(* IEC 61131-3 sources: TIA2AX/tests/test_projects/expected/HW_2200330_V18/ST70_PLC, 6 files *)

(* ---- HwInputs.st ---- *)
TYPE
	HwInputs : STRUCT
		ST70_ET200SP_CM_4xIO_Link_1 AT %B100 : ARRAY[0..31] OF BYTE;
		ST70_ET200SP_DI_16x24VDC_ST_1 AT %B0 : WORD;
		ST70_ET200SP_DI_16x24VDC_ST_2 AT %B2 : WORD;
		ST70_ET200SP_DI_8x24VDC_ST_3 AT %B4 : BYTE;
		ST70_ET200SP_DI_16x24VDC_ST_4 AT %B5 : WORD;
		ST70_1_DM260_PB_Acquisition_Status_1 AT %B1000 : ARRAY[0..2] OF BYTE;
		ST70_1_DM260_PB_Results_Status_1 AT %B1003 : BYTE;
		ST70_1_DM260_PB_Soft_Event_Control_1 AT %B1004 : BYTE;
		ST70_1_DM260_PB_Result_Data_64_bytes_1 AT %B1010 : ARRAY[0..71] OF BYTE;
		ST70_2_DM260_PB_Acquisition_Status_1 AT %B2000 : ARRAY[0..2] OF BYTE;
		ST70_2_DM260_PB_Results_Status_1 AT %B2003 : BYTE;
		ST70_2_DM260_PB_Soft_Event_Control_1 AT %B2004 : BYTE;
		ST70_2_DM260_PB_Result_Data_64_bytes_1 AT %B2010 : ARRAY[0..71] OF BYTE;
		ST70_3_DM260_PB_Acquisition_Status_1 AT %B3000 : ARRAY[0..2] OF BYTE;
		ST70_3_DM260_PB_Results_Status_1 AT %B3003 : BYTE;
		ST70_3_DM260_PB_Soft_Event_Control_1 AT %B3004 : BYTE;
		ST70_3_DM260_PB_Result_Data_64_bytes_1 AT %B3010 : ARRAY[0..71] OF BYTE;
		ST70_1_DM260_EB_Acquisition_Status_1 AT %B1200 : ARRAY[0..2] OF BYTE;
		ST70_1_DM260_EB_Results_Status_1 AT %B1203 : BYTE;
		ST70_1_DM260_EB_Soft_Event_Control_1 AT %B1204 : BYTE;
		ST70_1_DM260_EB_Result_Data_64_bytes_1 AT %B1210 : ARRAY[0..71] OF BYTE;
		ST70_2_DM260_EB_Acquisition_Status_1 AT %B2200 : ARRAY[0..2] OF BYTE;
		ST70_2_DM260_EB_Results_Status_1 AT %B2203 : BYTE;
		ST70_2_DM260_EB_Soft_Event_Control_1 AT %B2204 : BYTE;
		ST70_2_DM260_EB_Result_Data_64_bytes_1 AT %B2210 : ARRAY[0..71] OF BYTE;
		ST70_3_DM260_EB_Acquisition_Status_1 AT %B3200 : ARRAY[0..2] OF BYTE;
		ST70_3_DM260_EB_Results_Status_1 AT %B3203 : BYTE;
		ST70_3_DM260_EB_Soft_Event_Control_1 AT %B3204 : BYTE;
		ST70_3_DM260_EB_Result_Data_64_bytes_1 AT %B3210 : ARRAY[0..71] OF BYTE;
	END_STRUCT;
END_TYPE

(* ---- HwOutputs.st ---- *)
TYPE
	HwOutputs : STRUCT
		ST70_ET200SP_CM_4xIO_Link_1 AT %B100 : ARRAY[0..31] OF BYTE;
		ST70_ET200SP_DQ_16x24VDC_0_5A_ST_1 AT %B0 : WORD;
		ST70_ET200SP_DQ_16x24VDC_0_5A_ST_2 AT %B2 : WORD;
		ST70_ET200SP_DQ_16x24VDC_0_5A_ST_3 AT %B4 : WORD;
		ST70_CPX_MPA1S_VMPA1_FB_EMS_8_8DO_1 AT %B200 : BYTE;
		ST70_CPX_MPA1S_VMPA1_FB_EMS_8_8DO_2 AT %B201 : BYTE;
		ST70_CPX_MPA1S_VMPA1_FB_EMS_8_8DO_3 AT %B202 : BYTE;
		ST70_CPX_MPA2S_VMPA2_FB_EMS_4_4DO_1 AT %B6 : BYTE;
		ST70_CPX_MPA1G_VMPA1_FB_EMG_8_8DO_3 AT %B204 : BYTE;
		ST70_1_DM260_PB_Acquisition_Control_1 AT %B1000 : BYTE;
		ST70_1_DM260_PB_Results_Control_1 AT %B1003 : BYTE;
		ST70_1_DM260_PB_Soft_Event_Control_1 AT %B1004 : BYTE;
		ST70_1_DM260_PB_User_Data_64_bytes_1 AT %B1010 : ARRAY[0..67] OF BYTE;
		ST70_2_DM260_PB_Acquisition_Control_1 AT %B2000 : BYTE;
		ST70_2_DM260_PB_Results_Control_1 AT %B2003 : BYTE;
		ST70_2_DM260_PB_Soft_Event_Control_1 AT %B2004 : BYTE;
		ST70_2_DM260_PB_User_Data_64_bytes_1 AT %B2010 : ARRAY[0..67] OF BYTE;
		ST70_3_DM260_PB_Acquisition_Control_1 AT %B3000 : BYTE;
		ST70_3_DM260_PB_Results_Control_1 AT %B3003 : BYTE;
		ST70_3_DM260_PB_Soft_Event_Control_1 AT %B3004 : BYTE;
		ST70_3_DM260_PB_User_Data_64_bytes_1 AT %B3010 : ARRAY[0..67] OF BYTE;
		ST70_1_DM260_EB_Acquisition_Control_1 AT %B1200 : BYTE;
		ST70_1_DM260_EB_Results_Control_1 AT %B1203 : BYTE;
		ST70_1_DM260_EB_Soft_Event_Control_1 AT %B1204 : BYTE;
		ST70_1_DM260_EB_User_Data_64_bytes_1 AT %B1210 : ARRAY[0..67] OF BYTE;
		ST70_2_DM260_EB_Acquisition_Control_1 AT %B2200 : BYTE;
		ST70_2_DM260_EB_Results_Control_1 AT %B2203 : BYTE;
		ST70_2_DM260_EB_Soft_Event_Control_1 AT %B2204 : BYTE;
		ST70_2_DM260_EB_User_Data_64_bytes_1 AT %B2210 : ARRAY[0..67] OF BYTE;
		ST70_3_DM260_EB_Acquisition_Control_1 AT %B3200 : BYTE;
		ST70_3_DM260_EB_Results_Control_1 AT %B3203 : BYTE;
		ST70_3_DM260_EB_Soft_Event_Control_1 AT %B3204 : BYTE;
		ST70_3_DM260_EB_User_Data_64_bytes_1 AT %B3210 : ARRAY[0..67] OF BYTE;
	END_STRUCT;
END_TYPE

(* ---- PlcInputs.st ---- *)
TYPE
	PlcInputs : STRUCT
		ST70_ET200SP_CM_4xIO_Link_1 : ARRAY[0..31] OF BYTE;
		ST70_ET200SP_DI_16x24VDC_ST_1 : WORD;
		ST70_ET200SP_DI_16x24VDC_ST_2 : WORD;
		ST70_ET200SP_DI_8x24VDC_ST_3 : BYTE;
		ST70_ET200SP_DI_16x24VDC_ST_4 : WORD;
		ST70_1_DM260_PB_Acquisition_Status_1 : ARRAY[0..2] OF BYTE;
		ST70_1_DM260_PB_Results_Status_1 : BYTE;
		ST70_1_DM260_PB_Soft_Event_Control_1 : BYTE;
		ST70_1_DM260_PB_Result_Data_64_bytes_1 : ARRAY[0..71] OF BYTE;
		ST70_2_DM260_PB_Acquisition_Status_1 : ARRAY[0..2] OF BYTE;
		ST70_2_DM260_PB_Results_Status_1 : BYTE;
		ST70_2_DM260_PB_Soft_Event_Control_1 : BYTE;
		ST70_2_DM260_PB_Result_Data_64_bytes_1 : ARRAY[0..71] OF BYTE;
		ST70_3_DM260_PB_Acquisition_Status_1 : ARRAY[0..2] OF BYTE;
		ST70_3_DM260_PB_Results_Status_1 : BYTE;
		ST70_3_DM260_PB_Soft_Event_Control_1 : BYTE;
		ST70_3_DM260_PB_Result_Data_64_bytes_1 : ARRAY[0..71] OF BYTE;
		ST70_1_DM260_EB_Acquisition_Status_1 : ARRAY[0..2] OF BYTE;
		ST70_1_DM260_EB_Results_Status_1 : BYTE;
		ST70_1_DM260_EB_Soft_Event_Control_1 : BYTE;
		ST70_1_DM260_EB_Result_Data_64_bytes_1 : ARRAY[0..71] OF BYTE;
		ST70_2_DM260_EB_Acquisition_Status_1 : ARRAY[0..2] OF BYTE;
		ST70_2_DM260_EB_Results_Status_1 : BYTE;
		ST70_2_DM260_EB_Soft_Event_Control_1 : BYTE;
		ST70_2_DM260_EB_Result_Data_64_bytes_1 : ARRAY[0..71] OF BYTE;
		ST70_3_DM260_EB_Acquisition_Status_1 : ARRAY[0..2] OF BYTE;
		ST70_3_DM260_EB_Results_Status_1 : BYTE;
		ST70_3_DM260_EB_Soft_Event_Control_1 : BYTE;
		ST70_3_DM260_EB_Result_Data_64_bytes_1 : ARRAY[0..71] OF BYTE;
	END_STRUCT;
END_TYPE

(* ---- PlcOutputs.st ---- *)
TYPE
	PlcOutputs : STRUCT
		ST70_ET200SP_CM_4xIO_Link_1 : ARRAY[0..31] OF BYTE;
		ST70_ET200SP_DQ_16x24VDC_0_5A_ST_1 : WORD;
		ST70_ET200SP_DQ_16x24VDC_0_5A_ST_2 : WORD;
		ST70_ET200SP_DQ_16x24VDC_0_5A_ST_3 : WORD;
		ST70_CPX_MPA1S_VMPA1_FB_EMS_8_8DO_1 : BYTE;
		ST70_CPX_MPA1S_VMPA1_FB_EMS_8_8DO_2 : BYTE;
		ST70_CPX_MPA1S_VMPA1_FB_EMS_8_8DO_3 : BYTE;
		ST70_CPX_MPA2S_VMPA2_FB_EMS_4_4DO_1 : BYTE;
		ST70_CPX_MPA1G_VMPA1_FB_EMG_8_8DO_3 : BYTE;
		ST70_1_DM260_PB_Acquisition_Control_1 : BYTE;
		ST70_1_DM260_PB_Results_Control_1 : BYTE;
		ST70_1_DM260_PB_Soft_Event_Control_1 : BYTE;
		ST70_1_DM260_PB_User_Data_64_bytes_1 : ARRAY[0..67] OF BYTE;
		ST70_2_DM260_PB_Acquisition_Control_1 : BYTE;
		ST70_2_DM260_PB_Results_Control_1 : BYTE;
		ST70_2_DM260_PB_Soft_Event_Control_1 : BYTE;
		ST70_2_DM260_PB_User_Data_64_bytes_1 : ARRAY[0..67] OF BYTE;
		ST70_3_DM260_PB_Acquisition_Control_1 : BYTE;
		ST70_3_DM260_PB_Results_Control_1 : BYTE;
		ST70_3_DM260_PB_Soft_Event_Control_1 : BYTE;
		ST70_3_DM260_PB_User_Data_64_bytes_1 : ARRAY[0..67] OF BYTE;
		ST70_1_DM260_EB_Acquisition_Control_1 : BYTE;
		ST70_1_DM260_EB_Results_Control_1 : BYTE;
		ST70_1_DM260_EB_Soft_Event_Control_1 : BYTE;
		ST70_1_DM260_EB_User_Data_64_bytes_1 : ARRAY[0..67] OF BYTE;
		ST70_2_DM260_EB_Acquisition_Control_1 : BYTE;
		ST70_2_DM260_EB_Results_Control_1 : BYTE;
		ST70_2_DM260_EB_Soft_Event_Control_1 : BYTE;
		ST70_2_DM260_EB_User_Data_64_bytes_1 : ARRAY[0..67] OF BYTE;
		ST70_3_DM260_EB_Acquisition_Control_1 : BYTE;
		ST70_3_DM260_EB_Results_Control_1 : BYTE;
		ST70_3_DM260_EB_Soft_Event_Control_1 : BYTE;
		ST70_3_DM260_EB_User_Data_64_bytes_1 : ARRAY[0..67] OF BYTE;
	END_STRUCT;
END_TYPE

(* ---- CopyInputs.st ---- *)
FUNCTION CopyInputs
	VAR_EXTERNAL
		HwInputs : HwInputs;
		PlcInputs : PlcInputs;
	END_VAR
	PlcInputs.ST70_ET200SP_CM_4xIO_Link_1[0] := HwInputs.ST70_ET200SP_CM_4xIO_Link_1[0];
	PlcInputs.ST70_ET200SP_CM_4xIO_Link_1[1] := HwInputs.ST70_ET200SP_CM_4xIO_Link_1[1];
	PlcInputs.ST70_ET200SP_CM_4xIO_Link_1[2] := HwInputs.ST70_ET200SP_CM_4xIO_Link_1[2];
	PlcInputs.ST70_ET200SP_CM_4xIO_Link_1[3] := HwInputs.ST70_ET200SP_CM_4xIO_Link_1[3];
	PlcInputs.ST70_ET200SP_CM_4xIO_Link_1[4] := HwInputs.ST70_ET200SP_CM_4xIO_Link_1[4];
	PlcInputs.ST70_ET200SP_CM_4xIO_Link_1[5] := HwInputs.ST70_ET200SP_CM_4xIO_Link_1[5];
	PlcInputs.ST70_ET200SP_CM_4xIO_Link_1[6] := HwInputs.ST70_ET200SP_CM_4xIO_Link_1[6];
	PlcInputs.ST70_ET200SP_CM_4xIO_Link_1[7] := HwInputs.ST70_ET200SP_CM_4xIO_Link_1[7];
	PlcInputs.ST70_ET200SP_CM_4xIO_Link_1[8] := HwInputs.ST70_ET200SP_CM_4xIO_Link_1[8];
	PlcInputs.ST70_ET200SP_CM_4xIO_Link_1[9] := HwInputs.ST70_ET200SP_CM_4xIO_Link_1[9];
	PlcInputs.ST70_ET200SP_CM_4xIO_Link_1[10] := HwInputs.ST70_ET200SP_CM_4xIO_Link_1[10];
	PlcInputs.ST70_ET200SP_CM_4xIO_Link_1[11] := HwInputs.ST70_ET200SP_CM_4xIO_Link_1[11];
	PlcInputs.ST70_ET200SP_CM_4xIO_Link_1[12] := HwInputs.ST70_ET200SP_CM_4xIO_Link_1[12];
	PlcInputs.ST70_ET200SP_CM_4xIO_Link_1[13] := HwInputs.ST70_ET200SP_CM_4xIO_Link_1[13];
	PlcInputs.ST70_ET200SP_CM_4xIO_Link_1[14] := HwInputs.ST70_ET200SP_CM_4xIO_Link_1[14];
	PlcInputs.ST70_ET200SP_CM_4xIO_Link_1[15] := HwInputs.ST70_ET200SP_CM_4xIO_Link_1[15];
	PlcInputs.ST70_ET200SP_CM_4xIO_Link_1[16] := HwInputs.ST70_ET200SP_CM_4xIO_Link_1[16];
	PlcInputs.ST70_ET200SP_CM_4xIO_Link_1[17] := HwInputs.ST70_ET200SP_CM_4xIO_Link_1[17];
	PlcInputs.ST70_ET200SP_CM_4xIO_Link_1[18] := HwInputs.ST70_ET200SP_CM_4xIO_Link_1[18];
	PlcInputs.ST70_ET200SP_CM_4xIO_Link_1[19] := HwInputs.ST70_ET200SP_CM_4xIO_Link_1[19];
	PlcInputs.ST70_ET200SP_CM_4xIO_Link_1[20] := HwInputs.ST70_ET200SP_CM_4xIO_Link_1[20];
	PlcInputs.ST70_ET200SP_CM_4xIO_Link_1[21] := HwInputs.ST70_ET200SP_CM_4xIO_Link_1[21];
	PlcInputs.ST70_ET200SP_CM_4xIO_Link_1[22] := HwInputs.ST70_ET200SP_CM_4xIO_Link_1[22];
	PlcInputs.ST70_ET200SP_CM_4xIO_Link_1[23] := HwInputs.ST70_ET200SP_CM_4xIO_Link_1[23];
	PlcInputs.ST70_ET200SP_CM_4xIO_Link_1[24] := HwInputs.ST70_ET200SP_CM_4xIO_Link_1[24];
	PlcInputs.ST70_ET200SP_CM_4xIO_Link_1[25] := HwInputs.ST70_ET200SP_CM_4xIO_Link_1[25];
	PlcInputs.ST70_ET200SP_CM_4xIO_Link_1[26] := HwInputs.ST70_ET200SP_CM_4xIO_Link_1[26];
	PlcInputs.ST70_ET200SP_CM_4xIO_Link_1[27] := HwInputs.ST70_ET200SP_CM_4xIO_Link_1[27];
	PlcInputs.ST70_ET200SP_CM_4xIO_Link_1[28] := HwInputs.ST70_ET200SP_CM_4xIO_Link_1[28];
	PlcInputs.ST70_ET200SP_CM_4xIO_Link_1[29] := HwInputs.ST70_ET200SP_CM_4xIO_Link_1[29];
	PlcInputs.ST70_ET200SP_CM_4xIO_Link_1[30] := HwInputs.ST70_ET200SP_CM_4xIO_Link_1[30];
	PlcInputs.ST70_ET200SP_CM_4xIO_Link_1[31] := HwInputs.ST70_ET200SP_CM_4xIO_Link_1[31];
	PlcInputs.ST70_ET200SP_DI_16x24VDC_ST_1 := HwInputs.ST70_ET200SP_DI_16x24VDC_ST_1;
	PlcInputs.ST70_ET200SP_DI_16x24VDC_ST_2 := HwInputs.ST70_ET200SP_DI_16x24VDC_ST_2;
	PlcInputs.ST70_ET200SP_DI_8x24VDC_ST_3 := HwInputs.ST70_ET200SP_DI_8x24VDC_ST_3;
	PlcInputs.ST70_ET200SP_DI_16x24VDC_ST_4 := HwInputs.ST70_ET200SP_DI_16x24VDC_ST_4;
	PlcInputs.ST70_1_DM260_PB_Acquisition_Status_1[0] := HwInputs.ST70_1_DM260_PB_Acquisition_Status_1[0];
	PlcInputs.ST70_1_DM260_PB_Acquisition_Status_1[1] := HwInputs.ST70_1_DM260_PB_Acquisition_Status_1[1];
	PlcInputs.ST70_1_DM260_PB_Acquisition_Status_1[2] := HwInputs.ST70_1_DM260_PB_Acquisition_Status_1[2];
	PlcInputs.ST70_1_DM260_PB_Results_Status_1 := HwInputs.ST70_1_DM260_PB_Results_Status_1;
	PlcInputs.ST70_1_DM260_PB_Soft_Event_Control_1 := HwInputs.ST70_1_DM260_PB_Soft_Event_Control_1;
	PlcInputs.ST70_1_DM260_PB_Result_Data_64_bytes_1[0] := HwInputs.ST70_1_DM260_PB_Result_Data_64_bytes_1[0];
	PlcInputs.ST70_1_DM260_PB_Result_Data_64_bytes_1[1] := HwInputs.ST70_1_DM260_PB_Result_Data_64_bytes_1[1];
	PlcInputs.ST70_1_DM260_PB_Result_Data_64_bytes_1[2] := HwInputs.ST70_1_DM260_PB_Result_Data_64_bytes_1[2];
	PlcInputs.ST70_1_DM260_PB_Result_Data_64_bytes_1[3] := HwInputs.ST70_1_DM260_PB_Result_Data_64_bytes_1[3];
	PlcInputs.ST70_1_DM260_PB_Result_Data_64_bytes_1[4] := HwInputs.ST70_1_DM260_PB_Result_Data_64_bytes_1[4];
	PlcInputs.ST70_1_DM260_PB_Result_Data_64_bytes_1[5] := HwInputs.ST70_1_DM260_PB_Result_Data_64_bytes_1[5];
	PlcInputs.ST70_1_DM260_PB_Result_Data_64_bytes_1[6] := HwInputs.ST70_1_DM260_PB_Result_Data_64_bytes_1[6];
	PlcInputs.ST70_1_DM260_PB_Result_Data_64_bytes_1[7] := HwInputs.ST70_1_DM260_PB_Result_Data_64_bytes_1[7];
	PlcInputs.ST70_1_DM260_PB_Result_Data_64_bytes_1[8] := HwInputs.ST70_1_DM260_PB_Result_Data_64_bytes_1[8];
	PlcInputs.ST70_1_DM260_PB_Result_Data_64_bytes_1[9] := HwInputs.ST70_1_DM260_PB_Result_Data_64_bytes_1[9];
	PlcInputs.ST70_1_DM260_PB_Result_Data_64_bytes_1[10] := HwInputs.ST70_1_DM260_PB_Result_Data_64_bytes_1[10];
	PlcInputs.ST70_1_DM260_PB_Result_Data_64_bytes_1[11] := HwInputs.ST70_1_DM260_PB_Result_Data_64_bytes_1[11];
	PlcInputs.ST70_1_DM260_PB_Result_Data_64_bytes_1[12] := HwInputs.ST70_1_DM260_PB_Result_Data_64_bytes_1[12];
	PlcInputs.ST70_1_DM260_PB_Result_Data_64_bytes_1[13] := HwInputs.ST70_1_DM260_PB_Result_Data_64_bytes_1[13];
	PlcInputs.ST70_1_DM260_PB_Result_Data_64_bytes_1[14] := HwInputs.ST70_1_DM260_PB_Result_Data_64_bytes_1[14];
	PlcInputs.ST70_1_DM260_PB_Result_Data_64_bytes_1[15] := HwInputs.ST70_1_DM260_PB_Result_Data_64_bytes_1[15];
	PlcInputs.ST70_1_DM260_PB_Result_Data_64_bytes_1[16] := HwInputs.ST70_1_DM260_PB_Result_Data_64_bytes_1[16];
	PlcInputs.ST70_1_DM260_PB_Result_Data_64_bytes_1[17] := HwInputs.ST70_1_DM260_PB_Result_Data_64_bytes_1[17];
	PlcInputs.ST70_1_DM260_PB_Result_Data_64_bytes_1[18] := HwInputs.ST70_1_DM260_PB_Result_Data_64_bytes_1[18];
	PlcInputs.ST70_1_DM260_PB_Result_Data_64_bytes_1[19] := HwInputs.ST70_1_DM260_PB_Result_Data_64_bytes_1[19];
	PlcInputs.ST70_1_DM260_PB_Result_Data_64_bytes_1[20] := HwInputs.ST70_1_DM260_PB_Result_Data_64_bytes_1[20];
	PlcInputs.ST70_1_DM260_PB_Result_Data_64_bytes_1[21] := HwInputs.ST70_1_DM260_PB_Result_Data_64_bytes_1[21];
	PlcInputs.ST70_1_DM260_PB_Result_Data_64_bytes_1[22] := HwInputs.ST70_1_DM260_PB_Result_Data_64_bytes_1[22];
	PlcInputs.ST70_1_DM260_PB_Result_Data_64_bytes_1[23] := HwInputs.ST70_1_DM260_PB_Result_Data_64_bytes_1[23];
	PlcInputs.ST70_1_DM260_PB_Result_Data_64_bytes_1[24] := HwInputs.ST70_1_DM260_PB_Result_Data_64_bytes_1[24];
	PlcInputs.ST70_1_DM260_PB_Result_Data_64_bytes_1[25] := HwInputs.ST70_1_DM260_PB_Result_Data_64_bytes_1[25];
	PlcInputs.ST70_1_DM260_PB_Result_Data_64_bytes_1[26] := HwInputs.ST70_1_DM260_PB_Result_Data_64_bytes_1[26];
	PlcInputs.ST70_1_DM260_PB_Result_Data_64_bytes_1[27] := HwInputs.ST70_1_DM260_PB_Result_Data_64_bytes_1[27];
	PlcInputs.ST70_1_DM260_PB_Result_Data_64_bytes_1[28] := HwInputs.ST70_1_DM260_PB_Result_Data_64_bytes_1[28];
	PlcInputs.ST70_1_DM260_PB_Result_Data_64_bytes_1[29] := HwInputs.ST70_1_DM260_PB_Result_Data_64_bytes_1[29];
	PlcInputs.ST70_1_DM260_PB_Result_Data_64_bytes_1[30] := HwInputs.ST70_1_DM260_PB_Result_Data_64_bytes_1[30];
	PlcInputs.ST70_1_DM260_PB_Result_Data_64_bytes_1[31] := HwInputs.ST70_1_DM260_PB_Result_Data_64_bytes_1[31];
	PlcInputs.ST70_1_DM260_PB_Result_Data_64_bytes_1[32] := HwInputs.ST70_1_DM260_PB_Result_Data_64_bytes_1[32];
	PlcInputs.ST70_1_DM260_PB_Result_Data_64_bytes_1[33] := HwInputs.ST70_1_DM260_PB_Result_Data_64_bytes_1[33];
	PlcInputs.ST70_1_DM260_PB_Result_Data_64_bytes_1[34] := HwInputs.ST70_1_DM260_PB_Result_Data_64_bytes_1[34];
	PlcInputs.ST70_1_DM260_PB_Result_Data_64_bytes_1[35] := HwInputs.ST70_1_DM260_PB_Result_Data_64_bytes_1[35];
	PlcInputs.ST70_1_DM260_PB_Result_Data_64_bytes_1[36] := HwInputs.ST70_1_DM260_PB_Result_Data_64_bytes_1[36];
	PlcInputs.ST70_1_DM260_PB_Result_Data_64_bytes_1[37] := HwInputs.ST70_1_DM260_PB_Result_Data_64_bytes_1[37];
	PlcInputs.ST70_1_DM260_PB_Result_Data_64_bytes_1[38] := HwInputs.ST70_1_DM260_PB_Result_Data_64_bytes_1[38];
	PlcInputs.ST70_1_DM260_PB_Result_Data_64_bytes_1[39] := HwInputs.ST70_1_DM260_PB_Result_Data_64_bytes_1[39];
	PlcInputs.ST70_1_DM260_PB_Result_Data_64_bytes_1[40] := HwInputs.ST70_1_DM260_PB_Result_Data_64_bytes_1[40];
	PlcInputs.ST70_1_DM260_PB_Result_Data_64_bytes_1[41] := HwInputs.ST70_1_DM260_PB_Result_Data_64_bytes_1[41];
	PlcInputs.ST70_1_DM260_PB_Result_Data_64_bytes_1[42] := HwInputs.ST70_1_DM260_PB_Result_Data_64_bytes_1[42];
	PlcInputs.ST70_1_DM260_PB_Result_Data_64_bytes_1[43] := HwInputs.ST70_1_DM260_PB_Result_Data_64_bytes_1[43];
	PlcInputs.ST70_1_DM260_PB_Result_Data_64_bytes_1[44] := HwInputs.ST70_1_DM260_PB_Result_Data_64_bytes_1[44];
	PlcInputs.ST70_1_DM260_PB_Result_Data_64_bytes_1[45] := HwInputs.ST70_1_DM260_PB_Result_Data_64_bytes_1[45];
	PlcInputs.ST70_1_DM260_PB_Result_Data_64_bytes_1[46] := HwInputs.ST70_1_DM260_PB_Result_Data_64_bytes_1[46];
	PlcInputs.ST70_1_DM260_PB_Result_Data_64_bytes_1[47] := HwInputs.ST70_1_DM260_PB_Result_Data_64_bytes_1[47];
	PlcInputs.ST70_1_DM260_PB_Result_Data_64_bytes_1[48] := HwInputs.ST70_1_DM260_PB_Result_Data_64_bytes_1[48];
	PlcInputs.ST70_1_DM260_PB_Result_Data_64_bytes_1[49] := HwInputs.ST70_1_DM260_PB_Result_Data_64_bytes_1[49];
	PlcInputs.ST70_1_DM260_PB_Result_Data_64_bytes_1[50] := HwInputs.ST70_1_DM260_PB_Result_Data_64_bytes_1[50];
	PlcInputs.ST70_1_DM260_PB_Result_Data_64_bytes_1[51] := HwInputs.ST70_1_DM260_PB_Result_Data_64_bytes_1[51];
	PlcInputs.ST70_1_DM260_PB_Result_Data_64_bytes_1[52] := HwInputs.ST70_1_DM260_PB_Result_Data_64_bytes_1[52];
	PlcInputs.ST70_1_DM260_PB_Result_Data_64_bytes_1[53] := HwInputs.ST70_1_DM260_PB_Result_Data_64_bytes_1[53];
	PlcInputs.ST70_1_DM260_PB_Result_Data_64_bytes_1[54] := HwInputs.ST70_1_DM260_PB_Result_Data_64_bytes_1[54];
	PlcInputs.ST70_1_DM260_PB_Result_Data_64_bytes_1[55] := HwInputs.ST70_1_DM260_PB_Result_Data_64_bytes_1[55];
	PlcInputs.ST70_1_DM260_PB_Result_Data_64_bytes_1[56] := HwInputs.ST70_1_DM260_PB_Result_Data_64_bytes_1[56];
	PlcInputs.ST70_1_DM260_PB_Result_Data_64_bytes_1[57] := HwInputs.ST70_1_DM260_PB_Result_Data_64_bytes_1[57];
	PlcInputs.ST70_1_DM260_PB_Result_Data_64_bytes_1[58] := HwInputs.ST70_1_DM260_PB_Result_Data_64_bytes_1[58];
	PlcInputs.ST70_1_DM260_PB_Result_Data_64_bytes_1[59] := HwInputs.ST70_1_DM260_PB_Result_Data_64_bytes_1[59];
	PlcInputs.ST70_1_DM260_PB_Result_Data_64_bytes_1[60] := HwInputs.ST70_1_DM260_PB_Result_Data_64_bytes_1[60];
	PlcInputs.ST70_1_DM260_PB_Result_Data_64_bytes_1[61] := HwInputs.ST70_1_DM260_PB_Result_Data_64_bytes_1[61];
	PlcInputs.ST70_1_DM260_PB_Result_Data_64_bytes_1[62] := HwInputs.ST70_1_DM260_PB_Result_Data_64_bytes_1[62];
	PlcInputs.ST70_1_DM260_PB_Result_Data_64_bytes_1[63] := HwInputs.ST70_1_DM260_PB_Result_Data_64_bytes_1[63];
	PlcInputs.ST70_1_DM260_PB_Result_Data_64_bytes_1[64] := HwInputs.ST70_1_DM260_PB_Result_Data_64_bytes_1[64];
	PlcInputs.ST70_1_DM260_PB_Result_Data_64_bytes_1[65] := HwInputs.ST70_1_DM260_PB_Result_Data_64_bytes_1[65];
	PlcInputs.ST70_1_DM260_PB_Result_Data_64_bytes_1[66] := HwInputs.ST70_1_DM260_PB_Result_Data_64_bytes_1[66];
	PlcInputs.ST70_1_DM260_PB_Result_Data_64_bytes_1[67] := HwInputs.ST70_1_DM260_PB_Result_Data_64_bytes_1[67];
	PlcInputs.ST70_1_DM260_PB_Result_Data_64_bytes_1[68] := HwInputs.ST70_1_DM260_PB_Result_Data_64_bytes_1[68];
	PlcInputs.ST70_1_DM260_PB_Result_Data_64_bytes_1[69] := HwInputs.ST70_1_DM260_PB_Result_Data_64_bytes_1[69];
	PlcInputs.ST70_1_DM260_PB_Result_Data_64_bytes_1[70] := HwInputs.ST70_1_DM260_PB_Result_Data_64_bytes_1[70];
	PlcInputs.ST70_1_DM260_PB_Result_Data_64_bytes_1[71] := HwInputs.ST70_1_DM260_PB_Result_Data_64_bytes_1[71];
	PlcInputs.ST70_2_DM260_PB_Acquisition_Status_1[0] := HwInputs.ST70_2_DM260_PB_Acquisition_Status_1[0];
	PlcInputs.ST70_2_DM260_PB_Acquisition_Status_1[1] := HwInputs.ST70_2_DM260_PB_Acquisition_Status_1[1];
	PlcInputs.ST70_2_DM260_PB_Acquisition_Status_1[2] := HwInputs.ST70_2_DM260_PB_Acquisition_Status_1[2];
	PlcInputs.ST70_2_DM260_PB_Results_Status_1 := HwInputs.ST70_2_DM260_PB_Results_Status_1;
	PlcInputs.ST70_2_DM260_PB_Soft_Event_Control_1 := HwInputs.ST70_2_DM260_PB_Soft_Event_Control_1;
	PlcInputs.ST70_2_DM260_PB_Result_Data_64_bytes_1[0] := HwInputs.ST70_2_DM260_PB_Result_Data_64_bytes_1[0];
	PlcInputs.ST70_2_DM260_PB_Result_Data_64_bytes_1[1] := HwInputs.ST70_2_DM260_PB_Result_Data_64_bytes_1[1];
	PlcInputs.ST70_2_DM260_PB_Result_Data_64_bytes_1[2] := HwInputs.ST70_2_DM260_PB_Result_Data_64_bytes_1[2];
	PlcInputs.ST70_2_DM260_PB_Result_Data_64_bytes_1[3] := HwInputs.ST70_2_DM260_PB_Result_Data_64_bytes_1[3];
	PlcInputs.ST70_2_DM260_PB_Result_Data_64_bytes_1[4] := HwInputs.ST70_2_DM260_PB_Result_Data_64_bytes_1[4];
	PlcInputs.ST70_2_DM260_PB_Result_Data_64_bytes_1[5] := HwInputs.ST70_2_DM260_PB_Result_Data_64_bytes_1[5];
	PlcInputs.ST70_2_DM260_PB_Result_Data_64_bytes_1[6] := HwInputs.ST70_2_DM260_PB_Result_Data_64_bytes_1[6];
	PlcInputs.ST70_2_DM260_PB_Result_Data_64_bytes_1[7] := HwInputs.ST70_2_DM260_PB_Result_Data_64_bytes_1[7];
	PlcInputs.ST70_2_DM260_PB_Result_Data_64_bytes_1[8] := HwInputs.ST70_2_DM260_PB_Result_Data_64_bytes_1[8];
	PlcInputs.ST70_2_DM260_PB_Result_Data_64_bytes_1[9] := HwInputs.ST70_2_DM260_PB_Result_Data_64_bytes_1[9];
	PlcInputs.ST70_2_DM260_PB_Result_Data_64_bytes_1[10] := HwInputs.ST70_2_DM260_PB_Result_Data_64_bytes_1[10];
	PlcInputs.ST70_2_DM260_PB_Result_Data_64_bytes_1[11] := HwInputs.ST70_2_DM260_PB_Result_Data_64_bytes_1[11];
	PlcInputs.ST70_2_DM260_PB_Result_Data_64_bytes_1[12] := HwInputs.ST70_2_DM260_PB_Result_Data_64_bytes_1[12];
	PlcInputs.ST70_2_DM260_PB_Result_Data_64_bytes_1[13] := HwInputs.ST70_2_DM260_PB_Result_Data_64_bytes_1[13];
	PlcInputs.ST70_2_DM260_PB_Result_Data_64_bytes_1[14] := HwInputs.ST70_2_DM260_PB_Result_Data_64_bytes_1[14];
	PlcInputs.ST70_2_DM260_PB_Result_Data_64_bytes_1[15] := HwInputs.ST70_2_DM260_PB_Result_Data_64_bytes_1[15];
	PlcInputs.ST70_2_DM260_PB_Result_Data_64_bytes_1[16] := HwInputs.ST70_2_DM260_PB_Result_Data_64_bytes_1[16];
	PlcInputs.ST70_2_DM260_PB_Result_Data_64_bytes_1[17] := HwInputs.ST70_2_DM260_PB_Result_Data_64_bytes_1[17];
	PlcInputs.ST70_2_DM260_PB_Result_Data_64_bytes_1[18] := HwInputs.ST70_2_DM260_PB_Result_Data_64_bytes_1[18];
	PlcInputs.ST70_2_DM260_PB_Result_Data_64_bytes_1[19] := HwInputs.ST70_2_DM260_PB_Result_Data_64_bytes_1[19];
	PlcInputs.ST70_2_DM260_PB_Result_Data_64_bytes_1[20] := HwInputs.ST70_2_DM260_PB_Result_Data_64_bytes_1[20];
	PlcInputs.ST70_2_DM260_PB_Result_Data_64_bytes_1[21] := HwInputs.ST70_2_DM260_PB_Result_Data_64_bytes_1[21];
	PlcInputs.ST70_2_DM260_PB_Result_Data_64_bytes_1[22] := HwInputs.ST70_2_DM260_PB_Result_Data_64_bytes_1[22];
	PlcInputs.ST70_2_DM260_PB_Result_Data_64_bytes_1[23] := HwInputs.ST70_2_DM260_PB_Result_Data_64_bytes_1[23];
	PlcInputs.ST70_2_DM260_PB_Result_Data_64_bytes_1[24] := HwInputs.ST70_2_DM260_PB_Result_Data_64_bytes_1[24];
	PlcInputs.ST70_2_DM260_PB_Result_Data_64_bytes_1[25] := HwInputs.ST70_2_DM260_PB_Result_Data_64_bytes_1[25];
	PlcInputs.ST70_2_DM260_PB_Result_Data_64_bytes_1[26] := HwInputs.ST70_2_DM260_PB_Result_Data_64_bytes_1[26];
	PlcInputs.ST70_2_DM260_PB_Result_Data_64_bytes_1[27] := HwInputs.ST70_2_DM260_PB_Result_Data_64_bytes_1[27];
	PlcInputs.ST70_2_DM260_PB_Result_Data_64_bytes_1[28] := HwInputs.ST70_2_DM260_PB_Result_Data_64_bytes_1[28];
	PlcInputs.ST70_2_DM260_PB_Result_Data_64_bytes_1[29] := HwInputs.ST70_2_DM260_PB_Result_Data_64_bytes_1[29];
	PlcInputs.ST70_2_DM260_PB_Result_Data_64_bytes_1[30] := HwInputs.ST70_2_DM260_PB_Result_Data_64_bytes_1[30];
	PlcInputs.ST70_2_DM260_PB_Result_Data_64_bytes_1[31] := HwInputs.ST70_2_DM260_PB_Result_Data_64_bytes_1[31];
	PlcInputs.ST70_2_DM260_PB_Result_Data_64_bytes_1[32] := HwInputs.ST70_2_DM260_PB_Result_Data_64_bytes_1[32];
	PlcInputs.ST70_2_DM260_PB_Result_Data_64_bytes_1[33] := HwInputs.ST70_2_DM260_PB_Result_Data_64_bytes_1[33];
	PlcInputs.ST70_2_DM260_PB_Result_Data_64_bytes_1[34] := HwInputs.ST70_2_DM260_PB_Result_Data_64_bytes_1[34];
	PlcInputs.ST70_2_DM260_PB_Result_Data_64_bytes_1[35] := HwInputs.ST70_2_DM260_PB_Result_Data_64_bytes_1[35];
	PlcInputs.ST70_2_DM260_PB_Result_Data_64_bytes_1[36] := HwInputs.ST70_2_DM260_PB_Result_Data_64_bytes_1[36];
	PlcInputs.ST70_2_DM260_PB_Result_Data_64_bytes_1[37] := HwInputs.ST70_2_DM260_PB_Result_Data_64_bytes_1[37];
	PlcInputs.ST70_2_DM260_PB_Result_Data_64_bytes_1[38] := HwInputs.ST70_2_DM260_PB_Result_Data_64_bytes_1[38];
	PlcInputs.ST70_2_DM260_PB_Result_Data_64_bytes_1[39] := HwInputs.ST70_2_DM260_PB_Result_Data_64_bytes_1[39];
	PlcInputs.ST70_2_DM260_PB_Result_Data_64_bytes_1[40] := HwInputs.ST70_2_DM260_PB_Result_Data_64_bytes_1[40];
	PlcInputs.ST70_2_DM260_PB_Result_Data_64_bytes_1[41] := HwInputs.ST70_2_DM260_PB_Result_Data_64_bytes_1[41];
	PlcInputs.ST70_2_DM260_PB_Result_Data_64_bytes_1[42] := HwInputs.ST70_2_DM260_PB_Result_Data_64_bytes_1[42];
	PlcInputs.ST70_2_DM260_PB_Result_Data_64_bytes_1[43] := HwInputs.ST70_2_DM260_PB_Result_Data_64_bytes_1[43];
	PlcInputs.ST70_2_DM260_PB_Result_Data_64_bytes_1[44] := HwInputs.ST70_2_DM260_PB_Result_Data_64_bytes_1[44];
	PlcInputs.ST70_2_DM260_PB_Result_Data_64_bytes_1[45] := HwInputs.ST70_2_DM260_PB_Result_Data_64_bytes_1[45];
	PlcInputs.ST70_2_DM260_PB_Result_Data_64_bytes_1[46] := HwInputs.ST70_2_DM260_PB_Result_Data_64_bytes_1[46];
	PlcInputs.ST70_2_DM260_PB_Result_Data_64_bytes_1[47] := HwInputs.ST70_2_DM260_PB_Result_Data_64_bytes_1[47];
	PlcInputs.ST70_2_DM260_PB_Result_Data_64_bytes_1[48] := HwInputs.ST70_2_DM260_PB_Result_Data_64_bytes_1[48];
	PlcInputs.ST70_2_DM260_PB_Result_Data_64_bytes_1[49] := HwInputs.ST70_2_DM260_PB_Result_Data_64_bytes_1[49];
	PlcInputs.ST70_2_DM260_PB_Result_Data_64_bytes_1[50] := HwInputs.ST70_2_DM260_PB_Result_Data_64_bytes_1[50];
	PlcInputs.ST70_2_DM260_PB_Result_Data_64_bytes_1[51] := HwInputs.ST70_2_DM260_PB_Result_Data_64_bytes_1[51];
	PlcInputs.ST70_2_DM260_PB_Result_Data_64_bytes_1[52] := HwInputs.ST70_2_DM260_PB_Result_Data_64_bytes_1[52];
	PlcInputs.ST70_2_DM260_PB_Result_Data_64_bytes_1[53] := HwInputs.ST70_2_DM260_PB_Result_Data_64_bytes_1[53];
	PlcInputs.ST70_2_DM260_PB_Result_Data_64_bytes_1[54] := HwInputs.ST70_2_DM260_PB_Result_Data_64_bytes_1[54];
	PlcInputs.ST70_2_DM260_PB_Result_Data_64_bytes_1[55] := HwInputs.ST70_2_DM260_PB_Result_Data_64_bytes_1[55];
	PlcInputs.ST70_2_DM260_PB_Result_Data_64_bytes_1[56] := HwInputs.ST70_2_DM260_PB_Result_Data_64_bytes_1[56];
	PlcInputs.ST70_2_DM260_PB_Result_Data_64_bytes_1[57] := HwInputs.ST70_2_DM260_PB_Result_Data_64_bytes_1[57];
	PlcInputs.ST70_2_DM260_PB_Result_Data_64_bytes_1[58] := HwInputs.ST70_2_DM260_PB_Result_Data_64_bytes_1[58];
	PlcInputs.ST70_2_DM260_PB_Result_Data_64_bytes_1[59] := HwInputs.ST70_2_DM260_PB_Result_Data_64_bytes_1[59];
	PlcInputs.ST70_2_DM260_PB_Result_Data_64_bytes_1[60] := HwInputs.ST70_2_DM260_PB_Result_Data_64_bytes_1[60];
	PlcInputs.ST70_2_DM260_PB_Result_Data_64_bytes_1[61] := HwInputs.ST70_2_DM260_PB_Result_Data_64_bytes_1[61];
	PlcInputs.ST70_2_DM260_PB_Result_Data_64_bytes_1[62] := HwInputs.ST70_2_DM260_PB_Result_Data_64_bytes_1[62];
	PlcInputs.ST70_2_DM260_PB_Result_Data_64_bytes_1[63] := HwInputs.ST70_2_DM260_PB_Result_Data_64_bytes_1[63];
	PlcInputs.ST70_2_DM260_PB_Result_Data_64_bytes_1[64] := HwInputs.ST70_2_DM260_PB_Result_Data_64_bytes_1[64];
	PlcInputs.ST70_2_DM260_PB_Result_Data_64_bytes_1[65] := HwInputs.ST70_2_DM260_PB_Result_Data_64_bytes_1[65];
	PlcInputs.ST70_2_DM260_PB_Result_Data_64_bytes_1[66] := HwInputs.ST70_2_DM260_PB_Result_Data_64_bytes_1[66];
	PlcInputs.ST70_2_DM260_PB_Result_Data_64_bytes_1[67] := HwInputs.ST70_2_DM260_PB_Result_Data_64_bytes_1[67];
	PlcInputs.ST70_2_DM260_PB_Result_Data_64_bytes_1[68] := HwInputs.ST70_2_DM260_PB_Result_Data_64_bytes_1[68];
	PlcInputs.ST70_2_DM260_PB_Result_Data_64_bytes_1[69] := HwInputs.ST70_2_DM260_PB_Result_Data_64_bytes_1[69];
	PlcInputs.ST70_2_DM260_PB_Result_Data_64_bytes_1[70] := HwInputs.ST70_2_DM260_PB_Result_Data_64_bytes_1[70];
	PlcInputs.ST70_2_DM260_PB_Result_Data_64_bytes_1[71] := HwInputs.ST70_2_DM260_PB_Result_Data_64_bytes_1[71];
	PlcInputs.ST70_3_DM260_PB_Acquisition_Status_1[0] := HwInputs.ST70_3_DM260_PB_Acquisition_Status_1[0];
	PlcInputs.ST70_3_DM260_PB_Acquisition_Status_1[1] := HwInputs.ST70_3_DM260_PB_Acquisition_Status_1[1];
	PlcInputs.ST70_3_DM260_PB_Acquisition_Status_1[2] := HwInputs.ST70_3_DM260_PB_Acquisition_Status_1[2];
	PlcInputs.ST70_3_DM260_PB_Results_Status_1 := HwInputs.ST70_3_DM260_PB_Results_Status_1;
	PlcInputs.ST70_3_DM260_PB_Soft_Event_Control_1 := HwInputs.ST70_3_DM260_PB_Soft_Event_Control_1;
	PlcInputs.ST70_3_DM260_PB_Result_Data_64_bytes_1[0] := HwInputs.ST70_3_DM260_PB_Result_Data_64_bytes_1[0];
	PlcInputs.ST70_3_DM260_PB_Result_Data_64_bytes_1[1] := HwInputs.ST70_3_DM260_PB_Result_Data_64_bytes_1[1];
	PlcInputs.ST70_3_DM260_PB_Result_Data_64_bytes_1[2] := HwInputs.ST70_3_DM260_PB_Result_Data_64_bytes_1[2];
	PlcInputs.ST70_3_DM260_PB_Result_Data_64_bytes_1[3] := HwInputs.ST70_3_DM260_PB_Result_Data_64_bytes_1[3];
	PlcInputs.ST70_3_DM260_PB_Result_Data_64_bytes_1[4] := HwInputs.ST70_3_DM260_PB_Result_Data_64_bytes_1[4];
	PlcInputs.ST70_3_DM260_PB_Result_Data_64_bytes_1[5] := HwInputs.ST70_3_DM260_PB_Result_Data_64_bytes_1[5];
	PlcInputs.ST70_3_DM260_PB_Result_Data_64_bytes_1[6] := HwInputs.ST70_3_DM260_PB_Result_Data_64_bytes_1[6];
	PlcInputs.ST70_3_DM260_PB_Result_Data_64_bytes_1[7] := HwInputs.ST70_3_DM260_PB_Result_Data_64_bytes_1[7];
	PlcInputs.ST70_3_DM260_PB_Result_Data_64_bytes_1[8] := HwInputs.ST70_3_DM260_PB_Result_Data_64_bytes_1[8];
	PlcInputs.ST70_3_DM260_PB_Result_Data_64_bytes_1[9] := HwInputs.ST70_3_DM260_PB_Result_Data_64_bytes_1[9];
	PlcInputs.ST70_3_DM260_PB_Result_Data_64_bytes_1[10] := HwInputs.ST70_3_DM260_PB_Result_Data_64_bytes_1[10];
	PlcInputs.ST70_3_DM260_PB_Result_Data_64_bytes_1[11] := HwInputs.ST70_3_DM260_PB_Result_Data_64_bytes_1[11];
	PlcInputs.ST70_3_DM260_PB_Result_Data_64_bytes_1[12] := HwInputs.ST70_3_DM260_PB_Result_Data_64_bytes_1[12];
	PlcInputs.ST70_3_DM260_PB_Result_Data_64_bytes_1[13] := HwInputs.ST70_3_DM260_PB_Result_Data_64_bytes_1[13];
	PlcInputs.ST70_3_DM260_PB_Result_Data_64_bytes_1[14] := HwInputs.ST70_3_DM260_PB_Result_Data_64_bytes_1[14];
	PlcInputs.ST70_3_DM260_PB_Result_Data_64_bytes_1[15] := HwInputs.ST70_3_DM260_PB_Result_Data_64_bytes_1[15];
	PlcInputs.ST70_3_DM260_PB_Result_Data_64_bytes_1[16] := HwInputs.ST70_3_DM260_PB_Result_Data_64_bytes_1[16];
	PlcInputs.ST70_3_DM260_PB_Result_Data_64_bytes_1[17] := HwInputs.ST70_3_DM260_PB_Result_Data_64_bytes_1[17];
	PlcInputs.ST70_3_DM260_PB_Result_Data_64_bytes_1[18] := HwInputs.ST70_3_DM260_PB_Result_Data_64_bytes_1[18];
	PlcInputs.ST70_3_DM260_PB_Result_Data_64_bytes_1[19] := HwInputs.ST70_3_DM260_PB_Result_Data_64_bytes_1[19];
	PlcInputs.ST70_3_DM260_PB_Result_Data_64_bytes_1[20] := HwInputs.ST70_3_DM260_PB_Result_Data_64_bytes_1[20];
	PlcInputs.ST70_3_DM260_PB_Result_Data_64_bytes_1[21] := HwInputs.ST70_3_DM260_PB_Result_Data_64_bytes_1[21];
	PlcInputs.ST70_3_DM260_PB_Result_Data_64_bytes_1[22] := HwInputs.ST70_3_DM260_PB_Result_Data_64_bytes_1[22];
	PlcInputs.ST70_3_DM260_PB_Result_Data_64_bytes_1[23] := HwInputs.ST70_3_DM260_PB_Result_Data_64_bytes_1[23];
	PlcInputs.ST70_3_DM260_PB_Result_Data_64_bytes_1[24] := HwInputs.ST70_3_DM260_PB_Result_Data_64_bytes_1[24];
	PlcInputs.ST70_3_DM260_PB_Result_Data_64_bytes_1[25] := HwInputs.ST70_3_DM260_PB_Result_Data_64_bytes_1[25];
	PlcInputs.ST70_3_DM260_PB_Result_Data_64_bytes_1[26] := HwInputs.ST70_3_DM260_PB_Result_Data_64_bytes_1[26];
	PlcInputs.ST70_3_DM260_PB_Result_Data_64_bytes_1[27] := HwInputs.ST70_3_DM260_PB_Result_Data_64_bytes_1[27];
	PlcInputs.ST70_3_DM260_PB_Result_Data_64_bytes_1[28] := HwInputs.ST70_3_DM260_PB_Result_Data_64_bytes_1[28];
	PlcInputs.ST70_3_DM260_PB_Result_Data_64_bytes_1[29] := HwInputs.ST70_3_DM260_PB_Result_Data_64_bytes_1[29];
	PlcInputs.ST70_3_DM260_PB_Result_Data_64_bytes_1[30] := HwInputs.ST70_3_DM260_PB_Result_Data_64_bytes_1[30];
	PlcInputs.ST70_3_DM260_PB_Result_Data_64_bytes_1[31] := HwInputs.ST70_3_DM260_PB_Result_Data_64_bytes_1[31];
	PlcInputs.ST70_3_DM260_PB_Result_Data_64_bytes_1[32] := HwInputs.ST70_3_DM260_PB_Result_Data_64_bytes_1[32];
	PlcInputs.ST70_3_DM260_PB_Result_Data_64_bytes_1[33] := HwInputs.ST70_3_DM260_PB_Result_Data_64_bytes_1[33];
	PlcInputs.ST70_3_DM260_PB_Result_Data_64_bytes_1[34] := HwInputs.ST70_3_DM260_PB_Result_Data_64_bytes_1[34];
	PlcInputs.ST70_3_DM260_PB_Result_Data_64_bytes_1[35] := HwInputs.ST70_3_DM260_PB_Result_Data_64_bytes_1[35];
	PlcInputs.ST70_3_DM260_PB_Result_Data_64_bytes_1[36] := HwInputs.ST70_3_DM260_PB_Result_Data_64_bytes_1[36];
	PlcInputs.ST70_3_DM260_PB_Result_Data_64_bytes_1[37] := HwInputs.ST70_3_DM260_PB_Result_Data_64_bytes_1[37];
	PlcInputs.ST70_3_DM260_PB_Result_Data_64_bytes_1[38] := HwInputs.ST70_3_DM260_PB_Result_Data_64_bytes_1[38];
	PlcInputs.ST70_3_DM260_PB_Result_Data_64_bytes_1[39] := HwInputs.ST70_3_DM260_PB_Result_Data_64_bytes_1[39];
	PlcInputs.ST70_3_DM260_PB_Result_Data_64_bytes_1[40] := HwInputs.ST70_3_DM260_PB_Result_Data_64_bytes_1[40];
	PlcInputs.ST70_3_DM260_PB_Result_Data_64_bytes_1[41] := HwInputs.ST70_3_DM260_PB_Result_Data_64_bytes_1[41];
	PlcInputs.ST70_3_DM260_PB_Result_Data_64_bytes_1[42] := HwInputs.ST70_3_DM260_PB_Result_Data_64_bytes_1[42];
	PlcInputs.ST70_3_DM260_PB_Result_Data_64_bytes_1[43] := HwInputs.ST70_3_DM260_PB_Result_Data_64_bytes_1[43];
	PlcInputs.ST70_3_DM260_PB_Result_Data_64_bytes_1[44] := HwInputs.ST70_3_DM260_PB_Result_Data_64_bytes_1[44];
	PlcInputs.ST70_3_DM260_PB_Result_Data_64_bytes_1[45] := HwInputs.ST70_3_DM260_PB_Result_Data_64_bytes_1[45];
	PlcInputs.ST70_3_DM260_PB_Result_Data_64_bytes_1[46] := HwInputs.ST70_3_DM260_PB_Result_Data_64_bytes_1[46];
	PlcInputs.ST70_3_DM260_PB_Result_Data_64_bytes_1[47] := HwInputs.ST70_3_DM260_PB_Result_Data_64_bytes_1[47];
	PlcInputs.ST70_3_DM260_PB_Result_Data_64_bytes_1[48] := HwInputs.ST70_3_DM260_PB_Result_Data_64_bytes_1[48];
	PlcInputs.ST70_3_DM260_PB_Result_Data_64_bytes_1[49] := HwInputs.ST70_3_DM260_PB_Result_Data_64_bytes_1[49];
	PlcInputs.ST70_3_DM260_PB_Result_Data_64_bytes_1[50] := HwInputs.ST70_3_DM260_PB_Result_Data_64_bytes_1[50];
	PlcInputs.ST70_3_DM260_PB_Result_Data_64_bytes_1[51] := HwInputs.ST70_3_DM260_PB_Result_Data_64_bytes_1[51];
	PlcInputs.ST70_3_DM260_PB_Result_Data_64_bytes_1[52] := HwInputs.ST70_3_DM260_PB_Result_Data_64_bytes_1[52];
	PlcInputs.ST70_3_DM260_PB_Result_Data_64_bytes_1[53] := HwInputs.ST70_3_DM260_PB_Result_Data_64_bytes_1[53];
	PlcInputs.ST70_3_DM260_PB_Result_Data_64_bytes_1[54] := HwInputs.ST70_3_DM260_PB_Result_Data_64_bytes_1[54];
	PlcInputs.ST70_3_DM260_PB_Result_Data_64_bytes_1[55] := HwInputs.ST70_3_DM260_PB_Result_Data_64_bytes_1[55];
	PlcInputs.ST70_3_DM260_PB_Result_Data_64_bytes_1[56] := HwInputs.ST70_3_DM260_PB_Result_Data_64_bytes_1[56];
	PlcInputs.ST70_3_DM260_PB_Result_Data_64_bytes_1[57] := HwInputs.ST70_3_DM260_PB_Result_Data_64_bytes_1[57];
	PlcInputs.ST70_3_DM260_PB_Result_Data_64_bytes_1[58] := HwInputs.ST70_3_DM260_PB_Result_Data_64_bytes_1[58];
	PlcInputs.ST70_3_DM260_PB_Result_Data_64_bytes_1[59] := HwInputs.ST70_3_DM260_PB_Result_Data_64_bytes_1[59];
	PlcInputs.ST70_3_DM260_PB_Result_Data_64_bytes_1[60] := HwInputs.ST70_3_DM260_PB_Result_Data_64_bytes_1[60];
	PlcInputs.ST70_3_DM260_PB_Result_Data_64_bytes_1[61] := HwInputs.ST70_3_DM260_PB_Result_Data_64_bytes_1[61];
	PlcInputs.ST70_3_DM260_PB_Result_Data_64_bytes_1[62] := HwInputs.ST70_3_DM260_PB_Result_Data_64_bytes_1[62];
	PlcInputs.ST70_3_DM260_PB_Result_Data_64_bytes_1[63] := HwInputs.ST70_3_DM260_PB_Result_Data_64_bytes_1[63];
	PlcInputs.ST70_3_DM260_PB_Result_Data_64_bytes_1[64] := HwInputs.ST70_3_DM260_PB_Result_Data_64_bytes_1[64];
	PlcInputs.ST70_3_DM260_PB_Result_Data_64_bytes_1[65] := HwInputs.ST70_3_DM260_PB_Result_Data_64_bytes_1[65];
	PlcInputs.ST70_3_DM260_PB_Result_Data_64_bytes_1[66] := HwInputs.ST70_3_DM260_PB_Result_Data_64_bytes_1[66];
	PlcInputs.ST70_3_DM260_PB_Result_Data_64_bytes_1[67] := HwInputs.ST70_3_DM260_PB_Result_Data_64_bytes_1[67];
	PlcInputs.ST70_3_DM260_PB_Result_Data_64_bytes_1[68] := HwInputs.ST70_3_DM260_PB_Result_Data_64_bytes_1[68];
	PlcInputs.ST70_3_DM260_PB_Result_Data_64_bytes_1[69] := HwInputs.ST70_3_DM260_PB_Result_Data_64_bytes_1[69];
	PlcInputs.ST70_3_DM260_PB_Result_Data_64_bytes_1[70] := HwInputs.ST70_3_DM260_PB_Result_Data_64_bytes_1[70];
	PlcInputs.ST70_3_DM260_PB_Result_Data_64_bytes_1[71] := HwInputs.ST70_3_DM260_PB_Result_Data_64_bytes_1[71];
	PlcInputs.ST70_1_DM260_EB_Acquisition_Status_1[0] := HwInputs.ST70_1_DM260_EB_Acquisition_Status_1[0];
	PlcInputs.ST70_1_DM260_EB_Acquisition_Status_1[1] := HwInputs.ST70_1_DM260_EB_Acquisition_Status_1[1];
	PlcInputs.ST70_1_DM260_EB_Acquisition_Status_1[2] := HwInputs.ST70_1_DM260_EB_Acquisition_Status_1[2];
	PlcInputs.ST70_1_DM260_EB_Results_Status_1 := HwInputs.ST70_1_DM260_EB_Results_Status_1;
	PlcInputs.ST70_1_DM260_EB_Soft_Event_Control_1 := HwInputs.ST70_1_DM260_EB_Soft_Event_Control_1;
	PlcInputs.ST70_1_DM260_EB_Result_Data_64_bytes_1[0] := HwInputs.ST70_1_DM260_EB_Result_Data_64_bytes_1[0];
	PlcInputs.ST70_1_DM260_EB_Result_Data_64_bytes_1[1] := HwInputs.ST70_1_DM260_EB_Result_Data_64_bytes_1[1];
	PlcInputs.ST70_1_DM260_EB_Result_Data_64_bytes_1[2] := HwInputs.ST70_1_DM260_EB_Result_Data_64_bytes_1[2];
	PlcInputs.ST70_1_DM260_EB_Result_Data_64_bytes_1[3] := HwInputs.ST70_1_DM260_EB_Result_Data_64_bytes_1[3];
	PlcInputs.ST70_1_DM260_EB_Result_Data_64_bytes_1[4] := HwInputs.ST70_1_DM260_EB_Result_Data_64_bytes_1[4];
	PlcInputs.ST70_1_DM260_EB_Result_Data_64_bytes_1[5] := HwInputs.ST70_1_DM260_EB_Result_Data_64_bytes_1[5];
	PlcInputs.ST70_1_DM260_EB_Result_Data_64_bytes_1[6] := HwInputs.ST70_1_DM260_EB_Result_Data_64_bytes_1[6];
	PlcInputs.ST70_1_DM260_EB_Result_Data_64_bytes_1[7] := HwInputs.ST70_1_DM260_EB_Result_Data_64_bytes_1[7];
	PlcInputs.ST70_1_DM260_EB_Result_Data_64_bytes_1[8] := HwInputs.ST70_1_DM260_EB_Result_Data_64_bytes_1[8];
	PlcInputs.ST70_1_DM260_EB_Result_Data_64_bytes_1[9] := HwInputs.ST70_1_DM260_EB_Result_Data_64_bytes_1[9];
	PlcInputs.ST70_1_DM260_EB_Result_Data_64_bytes_1[10] := HwInputs.ST70_1_DM260_EB_Result_Data_64_bytes_1[10];
	PlcInputs.ST70_1_DM260_EB_Result_Data_64_bytes_1[11] := HwInputs.ST70_1_DM260_EB_Result_Data_64_bytes_1[11];
	PlcInputs.ST70_1_DM260_EB_Result_Data_64_bytes_1[12] := HwInputs.ST70_1_DM260_EB_Result_Data_64_bytes_1[12];
	PlcInputs.ST70_1_DM260_EB_Result_Data_64_bytes_1[13] := HwInputs.ST70_1_DM260_EB_Result_Data_64_bytes_1[13];
	PlcInputs.ST70_1_DM260_EB_Result_Data_64_bytes_1[14] := HwInputs.ST70_1_DM260_EB_Result_Data_64_bytes_1[14];
	PlcInputs.ST70_1_DM260_EB_Result_Data_64_bytes_1[15] := HwInputs.ST70_1_DM260_EB_Result_Data_64_bytes_1[15];
	PlcInputs.ST70_1_DM260_EB_Result_Data_64_bytes_1[16] := HwInputs.ST70_1_DM260_EB_Result_Data_64_bytes_1[16];
	PlcInputs.ST70_1_DM260_EB_Result_Data_64_bytes_1[17] := HwInputs.ST70_1_DM260_EB_Result_Data_64_bytes_1[17];
	PlcInputs.ST70_1_DM260_EB_Result_Data_64_bytes_1[18] := HwInputs.ST70_1_DM260_EB_Result_Data_64_bytes_1[18];
	PlcInputs.ST70_1_DM260_EB_Result_Data_64_bytes_1[19] := HwInputs.ST70_1_DM260_EB_Result_Data_64_bytes_1[19];
	PlcInputs.ST70_1_DM260_EB_Result_Data_64_bytes_1[20] := HwInputs.ST70_1_DM260_EB_Result_Data_64_bytes_1[20];
	PlcInputs.ST70_1_DM260_EB_Result_Data_64_bytes_1[21] := HwInputs.ST70_1_DM260_EB_Result_Data_64_bytes_1[21];
	PlcInputs.ST70_1_DM260_EB_Result_Data_64_bytes_1[22] := HwInputs.ST70_1_DM260_EB_Result_Data_64_bytes_1[22];
	PlcInputs.ST70_1_DM260_EB_Result_Data_64_bytes_1[23] := HwInputs.ST70_1_DM260_EB_Result_Data_64_bytes_1[23];
	PlcInputs.ST70_1_DM260_EB_Result_Data_64_bytes_1[24] := HwInputs.ST70_1_DM260_EB_Result_Data_64_bytes_1[24];
	PlcInputs.ST70_1_DM260_EB_Result_Data_64_bytes_1[25] := HwInputs.ST70_1_DM260_EB_Result_Data_64_bytes_1[25];
	PlcInputs.ST70_1_DM260_EB_Result_Data_64_bytes_1[26] := HwInputs.ST70_1_DM260_EB_Result_Data_64_bytes_1[26];
	PlcInputs.ST70_1_DM260_EB_Result_Data_64_bytes_1[27] := HwInputs.ST70_1_DM260_EB_Result_Data_64_bytes_1[27];
	PlcInputs.ST70_1_DM260_EB_Result_Data_64_bytes_1[28] := HwInputs.ST70_1_DM260_EB_Result_Data_64_bytes_1[28];
	PlcInputs.ST70_1_DM260_EB_Result_Data_64_bytes_1[29] := HwInputs.ST70_1_DM260_EB_Result_Data_64_bytes_1[29];
	PlcInputs.ST70_1_DM260_EB_Result_Data_64_bytes_1[30] := HwInputs.ST70_1_DM260_EB_Result_Data_64_bytes_1[30];
	PlcInputs.ST70_1_DM260_EB_Result_Data_64_bytes_1[31] := HwInputs.ST70_1_DM260_EB_Result_Data_64_bytes_1[31];
	PlcInputs.ST70_1_DM260_EB_Result_Data_64_bytes_1[32] := HwInputs.ST70_1_DM260_EB_Result_Data_64_bytes_1[32];
	PlcInputs.ST70_1_DM260_EB_Result_Data_64_bytes_1[33] := HwInputs.ST70_1_DM260_EB_Result_Data_64_bytes_1[33];
	PlcInputs.ST70_1_DM260_EB_Result_Data_64_bytes_1[34] := HwInputs.ST70_1_DM260_EB_Result_Data_64_bytes_1[34];
	PlcInputs.ST70_1_DM260_EB_Result_Data_64_bytes_1[35] := HwInputs.ST70_1_DM260_EB_Result_Data_64_bytes_1[35];
	PlcInputs.ST70_1_DM260_EB_Result_Data_64_bytes_1[36] := HwInputs.ST70_1_DM260_EB_Result_Data_64_bytes_1[36];
	PlcInputs.ST70_1_DM260_EB_Result_Data_64_bytes_1[37] := HwInputs.ST70_1_DM260_EB_Result_Data_64_bytes_1[37];
	PlcInputs.ST70_1_DM260_EB_Result_Data_64_bytes_1[38] := HwInputs.ST70_1_DM260_EB_Result_Data_64_bytes_1[38];
	PlcInputs.ST70_1_DM260_EB_Result_Data_64_bytes_1[39] := HwInputs.ST70_1_DM260_EB_Result_Data_64_bytes_1[39];
	PlcInputs.ST70_1_DM260_EB_Result_Data_64_bytes_1[40] := HwInputs.ST70_1_DM260_EB_Result_Data_64_bytes_1[40];
	PlcInputs.ST70_1_DM260_EB_Result_Data_64_bytes_1[41] := HwInputs.ST70_1_DM260_EB_Result_Data_64_bytes_1[41];
	PlcInputs.ST70_1_DM260_EB_Result_Data_64_bytes_1[42] := HwInputs.ST70_1_DM260_EB_Result_Data_64_bytes_1[42];
	PlcInputs.ST70_1_DM260_EB_Result_Data_64_bytes_1[43] := HwInputs.ST70_1_DM260_EB_Result_Data_64_bytes_1[43];
	PlcInputs.ST70_1_DM260_EB_Result_Data_64_bytes_1[44] := HwInputs.ST70_1_DM260_EB_Result_Data_64_bytes_1[44];
	PlcInputs.ST70_1_DM260_EB_Result_Data_64_bytes_1[45] := HwInputs.ST70_1_DM260_EB_Result_Data_64_bytes_1[45];
	PlcInputs.ST70_1_DM260_EB_Result_Data_64_bytes_1[46] := HwInputs.ST70_1_DM260_EB_Result_Data_64_bytes_1[46];
	PlcInputs.ST70_1_DM260_EB_Result_Data_64_bytes_1[47] := HwInputs.ST70_1_DM260_EB_Result_Data_64_bytes_1[47];
	PlcInputs.ST70_1_DM260_EB_Result_Data_64_bytes_1[48] := HwInputs.ST70_1_DM260_EB_Result_Data_64_bytes_1[48];
	PlcInputs.ST70_1_DM260_EB_Result_Data_64_bytes_1[49] := HwInputs.ST70_1_DM260_EB_Result_Data_64_bytes_1[49];
	PlcInputs.ST70_1_DM260_EB_Result_Data_64_bytes_1[50] := HwInputs.ST70_1_DM260_EB_Result_Data_64_bytes_1[50];
	PlcInputs.ST70_1_DM260_EB_Result_Data_64_bytes_1[51] := HwInputs.ST70_1_DM260_EB_Result_Data_64_bytes_1[51];
	PlcInputs.ST70_1_DM260_EB_Result_Data_64_bytes_1[52] := HwInputs.ST70_1_DM260_EB_Result_Data_64_bytes_1[52];
	PlcInputs.ST70_1_DM260_EB_Result_Data_64_bytes_1[53] := HwInputs.ST70_1_DM260_EB_Result_Data_64_bytes_1[53];
	PlcInputs.ST70_1_DM260_EB_Result_Data_64_bytes_1[54] := HwInputs.ST70_1_DM260_EB_Result_Data_64_bytes_1[54];
	PlcInputs.ST70_1_DM260_EB_Result_Data_64_bytes_1[55] := HwInputs.ST70_1_DM260_EB_Result_Data_64_bytes_1[55];
	PlcInputs.ST70_1_DM260_EB_Result_Data_64_bytes_1[56] := HwInputs.ST70_1_DM260_EB_Result_Data_64_bytes_1[56];
	PlcInputs.ST70_1_DM260_EB_Result_Data_64_bytes_1[57] := HwInputs.ST70_1_DM260_EB_Result_Data_64_bytes_1[57];
	PlcInputs.ST70_1_DM260_EB_Result_Data_64_bytes_1[58] := HwInputs.ST70_1_DM260_EB_Result_Data_64_bytes_1[58];
	PlcInputs.ST70_1_DM260_EB_Result_Data_64_bytes_1[59] := HwInputs.ST70_1_DM260_EB_Result_Data_64_bytes_1[59];
	PlcInputs.ST70_1_DM260_EB_Result_Data_64_bytes_1[60] := HwInputs.ST70_1_DM260_EB_Result_Data_64_bytes_1[60];
	PlcInputs.ST70_1_DM260_EB_Result_Data_64_bytes_1[61] := HwInputs.ST70_1_DM260_EB_Result_Data_64_bytes_1[61];
	PlcInputs.ST70_1_DM260_EB_Result_Data_64_bytes_1[62] := HwInputs.ST70_1_DM260_EB_Result_Data_64_bytes_1[62];
	PlcInputs.ST70_1_DM260_EB_Result_Data_64_bytes_1[63] := HwInputs.ST70_1_DM260_EB_Result_Data_64_bytes_1[63];
	PlcInputs.ST70_1_DM260_EB_Result_Data_64_bytes_1[64] := HwInputs.ST70_1_DM260_EB_Result_Data_64_bytes_1[64];
	PlcInputs.ST70_1_DM260_EB_Result_Data_64_bytes_1[65] := HwInputs.ST70_1_DM260_EB_Result_Data_64_bytes_1[65];
	PlcInputs.ST70_1_DM260_EB_Result_Data_64_bytes_1[66] := HwInputs.ST70_1_DM260_EB_Result_Data_64_bytes_1[66];
	PlcInputs.ST70_1_DM260_EB_Result_Data_64_bytes_1[67] := HwInputs.ST70_1_DM260_EB_Result_Data_64_bytes_1[67];
	PlcInputs.ST70_1_DM260_EB_Result_Data_64_bytes_1[68] := HwInputs.ST70_1_DM260_EB_Result_Data_64_bytes_1[68];
	PlcInputs.ST70_1_DM260_EB_Result_Data_64_bytes_1[69] := HwInputs.ST70_1_DM260_EB_Result_Data_64_bytes_1[69];
	PlcInputs.ST70_1_DM260_EB_Result_Data_64_bytes_1[70] := HwInputs.ST70_1_DM260_EB_Result_Data_64_bytes_1[70];
	PlcInputs.ST70_1_DM260_EB_Result_Data_64_bytes_1[71] := HwInputs.ST70_1_DM260_EB_Result_Data_64_bytes_1[71];
	PlcInputs.ST70_2_DM260_EB_Acquisition_Status_1[0] := HwInputs.ST70_2_DM260_EB_Acquisition_Status_1[0];
	PlcInputs.ST70_2_DM260_EB_Acquisition_Status_1[1] := HwInputs.ST70_2_DM260_EB_Acquisition_Status_1[1];
	PlcInputs.ST70_2_DM260_EB_Acquisition_Status_1[2] := HwInputs.ST70_2_DM260_EB_Acquisition_Status_1[2];
	PlcInputs.ST70_2_DM260_EB_Results_Status_1 := HwInputs.ST70_2_DM260_EB_Results_Status_1;
	PlcInputs.ST70_2_DM260_EB_Soft_Event_Control_1 := HwInputs.ST70_2_DM260_EB_Soft_Event_Control_1;
	PlcInputs.ST70_2_DM260_EB_Result_Data_64_bytes_1[0] := HwInputs.ST70_2_DM260_EB_Result_Data_64_bytes_1[0];
	PlcInputs.ST70_2_DM260_EB_Result_Data_64_bytes_1[1] := HwInputs.ST70_2_DM260_EB_Result_Data_64_bytes_1[1];
	PlcInputs.ST70_2_DM260_EB_Result_Data_64_bytes_1[2] := HwInputs.ST70_2_DM260_EB_Result_Data_64_bytes_1[2];
	PlcInputs.ST70_2_DM260_EB_Result_Data_64_bytes_1[3] := HwInputs.ST70_2_DM260_EB_Result_Data_64_bytes_1[3];
	PlcInputs.ST70_2_DM260_EB_Result_Data_64_bytes_1[4] := HwInputs.ST70_2_DM260_EB_Result_Data_64_bytes_1[4];
	PlcInputs.ST70_2_DM260_EB_Result_Data_64_bytes_1[5] := HwInputs.ST70_2_DM260_EB_Result_Data_64_bytes_1[5];
	PlcInputs.ST70_2_DM260_EB_Result_Data_64_bytes_1[6] := HwInputs.ST70_2_DM260_EB_Result_Data_64_bytes_1[6];
	PlcInputs.ST70_2_DM260_EB_Result_Data_64_bytes_1[7] := HwInputs.ST70_2_DM260_EB_Result_Data_64_bytes_1[7];
	PlcInputs.ST70_2_DM260_EB_Result_Data_64_bytes_1[8] := HwInputs.ST70_2_DM260_EB_Result_Data_64_bytes_1[8];
	PlcInputs.ST70_2_DM260_EB_Result_Data_64_bytes_1[9] := HwInputs.ST70_2_DM260_EB_Result_Data_64_bytes_1[9];
	PlcInputs.ST70_2_DM260_EB_Result_Data_64_bytes_1[10] := HwInputs.ST70_2_DM260_EB_Result_Data_64_bytes_1[10];
	PlcInputs.ST70_2_DM260_EB_Result_Data_64_bytes_1[11] := HwInputs.ST70_2_DM260_EB_Result_Data_64_bytes_1[11];
	PlcInputs.ST70_2_DM260_EB_Result_Data_64_bytes_1[12] := HwInputs.ST70_2_DM260_EB_Result_Data_64_bytes_1[12];
	PlcInputs.ST70_2_DM260_EB_Result_Data_64_bytes_1[13] := HwInputs.ST70_2_DM260_EB_Result_Data_64_bytes_1[13];
	PlcInputs.ST70_2_DM260_EB_Result_Data_64_bytes_1[14] := HwInputs.ST70_2_DM260_EB_Result_Data_64_bytes_1[14];
	PlcInputs.ST70_2_DM260_EB_Result_Data_64_bytes_1[15] := HwInputs.ST70_2_DM260_EB_Result_Data_64_bytes_1[15];
	PlcInputs.ST70_2_DM260_EB_Result_Data_64_bytes_1[16] := HwInputs.ST70_2_DM260_EB_Result_Data_64_bytes_1[16];
	PlcInputs.ST70_2_DM260_EB_Result_Data_64_bytes_1[17] := HwInputs.ST70_2_DM260_EB_Result_Data_64_bytes_1[17];
	PlcInputs.ST70_2_DM260_EB_Result_Data_64_bytes_1[18] := HwInputs.ST70_2_DM260_EB_Result_Data_64_bytes_1[18];
	PlcInputs.ST70_2_DM260_EB_Result_Data_64_bytes_1[19] := HwInputs.ST70_2_DM260_EB_Result_Data_64_bytes_1[19];
	PlcInputs.ST70_2_DM260_EB_Result_Data_64_bytes_1[20] := HwInputs.ST70_2_DM260_EB_Result_Data_64_bytes_1[20];
	PlcInputs.ST70_2_DM260_EB_Result_Data_64_bytes_1[21] := HwInputs.ST70_2_DM260_EB_Result_Data_64_bytes_1[21];
	PlcInputs.ST70_2_DM260_EB_Result_Data_64_bytes_1[22] := HwInputs.ST70_2_DM260_EB_Result_Data_64_bytes_1[22];
	PlcInputs.ST70_2_DM260_EB_Result_Data_64_bytes_1[23] := HwInputs.ST70_2_DM260_EB_Result_Data_64_bytes_1[23];
	PlcInputs.ST70_2_DM260_EB_Result_Data_64_bytes_1[24] := HwInputs.ST70_2_DM260_EB_Result_Data_64_bytes_1[24];
	PlcInputs.ST70_2_DM260_EB_Result_Data_64_bytes_1[25] := HwInputs.ST70_2_DM260_EB_Result_Data_64_bytes_1[25];
	PlcInputs.ST70_2_DM260_EB_Result_Data_64_bytes_1[26] := HwInputs.ST70_2_DM260_EB_Result_Data_64_bytes_1[26];
	PlcInputs.ST70_2_DM260_EB_Result_Data_64_bytes_1[27] := HwInputs.ST70_2_DM260_EB_Result_Data_64_bytes_1[27];
	PlcInputs.ST70_2_DM260_EB_Result_Data_64_bytes_1[28] := HwInputs.ST70_2_DM260_EB_Result_Data_64_bytes_1[28];
	PlcInputs.ST70_2_DM260_EB_Result_Data_64_bytes_1[29] := HwInputs.ST70_2_DM260_EB_Result_Data_64_bytes_1[29];
	PlcInputs.ST70_2_DM260_EB_Result_Data_64_bytes_1[30] := HwInputs.ST70_2_DM260_EB_Result_Data_64_bytes_1[30];
	PlcInputs.ST70_2_DM260_EB_Result_Data_64_bytes_1[31] := HwInputs.ST70_2_DM260_EB_Result_Data_64_bytes_1[31];
	PlcInputs.ST70_2_DM260_EB_Result_Data_64_bytes_1[32] := HwInputs.ST70_2_DM260_EB_Result_Data_64_bytes_1[32];
	PlcInputs.ST70_2_DM260_EB_Result_Data_64_bytes_1[33] := HwInputs.ST70_2_DM260_EB_Result_Data_64_bytes_1[33];
	PlcInputs.ST70_2_DM260_EB_Result_Data_64_bytes_1[34] := HwInputs.ST70_2_DM260_EB_Result_Data_64_bytes_1[34];
	PlcInputs.ST70_2_DM260_EB_Result_Data_64_bytes_1[35] := HwInputs.ST70_2_DM260_EB_Result_Data_64_bytes_1[35];
	PlcInputs.ST70_2_DM260_EB_Result_Data_64_bytes_1[36] := HwInputs.ST70_2_DM260_EB_Result_Data_64_bytes_1[36];
	PlcInputs.ST70_2_DM260_EB_Result_Data_64_bytes_1[37] := HwInputs.ST70_2_DM260_EB_Result_Data_64_bytes_1[37];
	PlcInputs.ST70_2_DM260_EB_Result_Data_64_bytes_1[38] := HwInputs.ST70_2_DM260_EB_Result_Data_64_bytes_1[38];
	PlcInputs.ST70_2_DM260_EB_Result_Data_64_bytes_1[39] := HwInputs.ST70_2_DM260_EB_Result_Data_64_bytes_1[39];
	PlcInputs.ST70_2_DM260_EB_Result_Data_64_bytes_1[40] := HwInputs.ST70_2_DM260_EB_Result_Data_64_bytes_1[40];
	PlcInputs.ST70_2_DM260_EB_Result_Data_64_bytes_1[41] := HwInputs.ST70_2_DM260_EB_Result_Data_64_bytes_1[41];
	PlcInputs.ST70_2_DM260_EB_Result_Data_64_bytes_1[42] := HwInputs.ST70_2_DM260_EB_Result_Data_64_bytes_1[42];
	PlcInputs.ST70_2_DM260_EB_Result_Data_64_bytes_1[43] := HwInputs.ST70_2_DM260_EB_Result_Data_64_bytes_1[43];
	PlcInputs.ST70_2_DM260_EB_Result_Data_64_bytes_1[44] := HwInputs.ST70_2_DM260_EB_Result_Data_64_bytes_1[44];
	PlcInputs.ST70_2_DM260_EB_Result_Data_64_bytes_1[45] := HwInputs.ST70_2_DM260_EB_Result_Data_64_bytes_1[45];
	PlcInputs.ST70_2_DM260_EB_Result_Data_64_bytes_1[46] := HwInputs.ST70_2_DM260_EB_Result_Data_64_bytes_1[46];
	PlcInputs.ST70_2_DM260_EB_Result_Data_64_bytes_1[47] := HwInputs.ST70_2_DM260_EB_Result_Data_64_bytes_1[47];
	PlcInputs.ST70_2_DM260_EB_Result_Data_64_bytes_1[48] := HwInputs.ST70_2_DM260_EB_Result_Data_64_bytes_1[48];
	PlcInputs.ST70_2_DM260_EB_Result_Data_64_bytes_1[49] := HwInputs.ST70_2_DM260_EB_Result_Data_64_bytes_1[49];
	PlcInputs.ST70_2_DM260_EB_Result_Data_64_bytes_1[50] := HwInputs.ST70_2_DM260_EB_Result_Data_64_bytes_1[50];
	PlcInputs.ST70_2_DM260_EB_Result_Data_64_bytes_1[51] := HwInputs.ST70_2_DM260_EB_Result_Data_64_bytes_1[51];
	PlcInputs.ST70_2_DM260_EB_Result_Data_64_bytes_1[52] := HwInputs.ST70_2_DM260_EB_Result_Data_64_bytes_1[52];
	PlcInputs.ST70_2_DM260_EB_Result_Data_64_bytes_1[53] := HwInputs.ST70_2_DM260_EB_Result_Data_64_bytes_1[53];
	PlcInputs.ST70_2_DM260_EB_Result_Data_64_bytes_1[54] := HwInputs.ST70_2_DM260_EB_Result_Data_64_bytes_1[54];
	PlcInputs.ST70_2_DM260_EB_Result_Data_64_bytes_1[55] := HwInputs.ST70_2_DM260_EB_Result_Data_64_bytes_1[55];
	PlcInputs.ST70_2_DM260_EB_Result_Data_64_bytes_1[56] := HwInputs.ST70_2_DM260_EB_Result_Data_64_bytes_1[56];
	PlcInputs.ST70_2_DM260_EB_Result_Data_64_bytes_1[57] := HwInputs.ST70_2_DM260_EB_Result_Data_64_bytes_1[57];
	PlcInputs.ST70_2_DM260_EB_Result_Data_64_bytes_1[58] := HwInputs.ST70_2_DM260_EB_Result_Data_64_bytes_1[58];
	PlcInputs.ST70_2_DM260_EB_Result_Data_64_bytes_1[59] := HwInputs.ST70_2_DM260_EB_Result_Data_64_bytes_1[59];
	PlcInputs.ST70_2_DM260_EB_Result_Data_64_bytes_1[60] := HwInputs.ST70_2_DM260_EB_Result_Data_64_bytes_1[60];
	PlcInputs.ST70_2_DM260_EB_Result_Data_64_bytes_1[61] := HwInputs.ST70_2_DM260_EB_Result_Data_64_bytes_1[61];
	PlcInputs.ST70_2_DM260_EB_Result_Data_64_bytes_1[62] := HwInputs.ST70_2_DM260_EB_Result_Data_64_bytes_1[62];
	PlcInputs.ST70_2_DM260_EB_Result_Data_64_bytes_1[63] := HwInputs.ST70_2_DM260_EB_Result_Data_64_bytes_1[63];
	PlcInputs.ST70_2_DM260_EB_Result_Data_64_bytes_1[64] := HwInputs.ST70_2_DM260_EB_Result_Data_64_bytes_1[64];
	PlcInputs.ST70_2_DM260_EB_Result_Data_64_bytes_1[65] := HwInputs.ST70_2_DM260_EB_Result_Data_64_bytes_1[65];
	PlcInputs.ST70_2_DM260_EB_Result_Data_64_bytes_1[66] := HwInputs.ST70_2_DM260_EB_Result_Data_64_bytes_1[66];
	PlcInputs.ST70_2_DM260_EB_Result_Data_64_bytes_1[67] := HwInputs.ST70_2_DM260_EB_Result_Data_64_bytes_1[67];
	PlcInputs.ST70_2_DM260_EB_Result_Data_64_bytes_1[68] := HwInputs.ST70_2_DM260_EB_Result_Data_64_bytes_1[68];
	PlcInputs.ST70_2_DM260_EB_Result_Data_64_bytes_1[69] := HwInputs.ST70_2_DM260_EB_Result_Data_64_bytes_1[69];
	PlcInputs.ST70_2_DM260_EB_Result_Data_64_bytes_1[70] := HwInputs.ST70_2_DM260_EB_Result_Data_64_bytes_1[70];
	PlcInputs.ST70_2_DM260_EB_Result_Data_64_bytes_1[71] := HwInputs.ST70_2_DM260_EB_Result_Data_64_bytes_1[71];
	PlcInputs.ST70_3_DM260_EB_Acquisition_Status_1[0] := HwInputs.ST70_3_DM260_EB_Acquisition_Status_1[0];
	PlcInputs.ST70_3_DM260_EB_Acquisition_Status_1[1] := HwInputs.ST70_3_DM260_EB_Acquisition_Status_1[1];
	PlcInputs.ST70_3_DM260_EB_Acquisition_Status_1[2] := HwInputs.ST70_3_DM260_EB_Acquisition_Status_1[2];
	PlcInputs.ST70_3_DM260_EB_Results_Status_1 := HwInputs.ST70_3_DM260_EB_Results_Status_1;
	PlcInputs.ST70_3_DM260_EB_Soft_Event_Control_1 := HwInputs.ST70_3_DM260_EB_Soft_Event_Control_1;
	PlcInputs.ST70_3_DM260_EB_Result_Data_64_bytes_1[0] := HwInputs.ST70_3_DM260_EB_Result_Data_64_bytes_1[0];
	PlcInputs.ST70_3_DM260_EB_Result_Data_64_bytes_1[1] := HwInputs.ST70_3_DM260_EB_Result_Data_64_bytes_1[1];
	PlcInputs.ST70_3_DM260_EB_Result_Data_64_bytes_1[2] := HwInputs.ST70_3_DM260_EB_Result_Data_64_bytes_1[2];
	PlcInputs.ST70_3_DM260_EB_Result_Data_64_bytes_1[3] := HwInputs.ST70_3_DM260_EB_Result_Data_64_bytes_1[3];
	PlcInputs.ST70_3_DM260_EB_Result_Data_64_bytes_1[4] := HwInputs.ST70_3_DM260_EB_Result_Data_64_bytes_1[4];
	PlcInputs.ST70_3_DM260_EB_Result_Data_64_bytes_1[5] := HwInputs.ST70_3_DM260_EB_Result_Data_64_bytes_1[5];
	PlcInputs.ST70_3_DM260_EB_Result_Data_64_bytes_1[6] := HwInputs.ST70_3_DM260_EB_Result_Data_64_bytes_1[6];
	PlcInputs.ST70_3_DM260_EB_Result_Data_64_bytes_1[7] := HwInputs.ST70_3_DM260_EB_Result_Data_64_bytes_1[7];
	PlcInputs.ST70_3_DM260_EB_Result_Data_64_bytes_1[8] := HwInputs.ST70_3_DM260_EB_Result_Data_64_bytes_1[8];
	PlcInputs.ST70_3_DM260_EB_Result_Data_64_bytes_1[9] := HwInputs.ST70_3_DM260_EB_Result_Data_64_bytes_1[9];
	PlcInputs.ST70_3_DM260_EB_Result_Data_64_bytes_1[10] := HwInputs.ST70_3_DM260_EB_Result_Data_64_bytes_1[10];
	PlcInputs.ST70_3_DM260_EB_Result_Data_64_bytes_1[11] := HwInputs.ST70_3_DM260_EB_Result_Data_64_bytes_1[11];
	PlcInputs.ST70_3_DM260_EB_Result_Data_64_bytes_1[12] := HwInputs.ST70_3_DM260_EB_Result_Data_64_bytes_1[12];
	PlcInputs.ST70_3_DM260_EB_Result_Data_64_bytes_1[13] := HwInputs.ST70_3_DM260_EB_Result_Data_64_bytes_1[13];
	PlcInputs.ST70_3_DM260_EB_Result_Data_64_bytes_1[14] := HwInputs.ST70_3_DM260_EB_Result_Data_64_bytes_1[14];
	PlcInputs.ST70_3_DM260_EB_Result_Data_64_bytes_1[15] := HwInputs.ST70_3_DM260_EB_Result_Data_64_bytes_1[15];
	PlcInputs.ST70_3_DM260_EB_Result_Data_64_bytes_1[16] := HwInputs.ST70_3_DM260_EB_Result_Data_64_bytes_1[16];
	PlcInputs.ST70_3_DM260_EB_Result_Data_64_bytes_1[17] := HwInputs.ST70_3_DM260_EB_Result_Data_64_bytes_1[17];
	PlcInputs.ST70_3_DM260_EB_Result_Data_64_bytes_1[18] := HwInputs.ST70_3_DM260_EB_Result_Data_64_bytes_1[18];
	PlcInputs.ST70_3_DM260_EB_Result_Data_64_bytes_1[19] := HwInputs.ST70_3_DM260_EB_Result_Data_64_bytes_1[19];
	PlcInputs.ST70_3_DM260_EB_Result_Data_64_bytes_1[20] := HwInputs.ST70_3_DM260_EB_Result_Data_64_bytes_1[20];
	PlcInputs.ST70_3_DM260_EB_Result_Data_64_bytes_1[21] := HwInputs.ST70_3_DM260_EB_Result_Data_64_bytes_1[21];
	PlcInputs.ST70_3_DM260_EB_Result_Data_64_bytes_1[22] := HwInputs.ST70_3_DM260_EB_Result_Data_64_bytes_1[22];
	PlcInputs.ST70_3_DM260_EB_Result_Data_64_bytes_1[23] := HwInputs.ST70_3_DM260_EB_Result_Data_64_bytes_1[23];
	PlcInputs.ST70_3_DM260_EB_Result_Data_64_bytes_1[24] := HwInputs.ST70_3_DM260_EB_Result_Data_64_bytes_1[24];
	PlcInputs.ST70_3_DM260_EB_Result_Data_64_bytes_1[25] := HwInputs.ST70_3_DM260_EB_Result_Data_64_bytes_1[25];
	PlcInputs.ST70_3_DM260_EB_Result_Data_64_bytes_1[26] := HwInputs.ST70_3_DM260_EB_Result_Data_64_bytes_1[26];
	PlcInputs.ST70_3_DM260_EB_Result_Data_64_bytes_1[27] := HwInputs.ST70_3_DM260_EB_Result_Data_64_bytes_1[27];
	PlcInputs.ST70_3_DM260_EB_Result_Data_64_bytes_1[28] := HwInputs.ST70_3_DM260_EB_Result_Data_64_bytes_1[28];
	PlcInputs.ST70_3_DM260_EB_Result_Data_64_bytes_1[29] := HwInputs.ST70_3_DM260_EB_Result_Data_64_bytes_1[29];
	PlcInputs.ST70_3_DM260_EB_Result_Data_64_bytes_1[30] := HwInputs.ST70_3_DM260_EB_Result_Data_64_bytes_1[30];
	PlcInputs.ST70_3_DM260_EB_Result_Data_64_bytes_1[31] := HwInputs.ST70_3_DM260_EB_Result_Data_64_bytes_1[31];
	PlcInputs.ST70_3_DM260_EB_Result_Data_64_bytes_1[32] := HwInputs.ST70_3_DM260_EB_Result_Data_64_bytes_1[32];
	PlcInputs.ST70_3_DM260_EB_Result_Data_64_bytes_1[33] := HwInputs.ST70_3_DM260_EB_Result_Data_64_bytes_1[33];
	PlcInputs.ST70_3_DM260_EB_Result_Data_64_bytes_1[34] := HwInputs.ST70_3_DM260_EB_Result_Data_64_bytes_1[34];
	PlcInputs.ST70_3_DM260_EB_Result_Data_64_bytes_1[35] := HwInputs.ST70_3_DM260_EB_Result_Data_64_bytes_1[35];
	PlcInputs.ST70_3_DM260_EB_Result_Data_64_bytes_1[36] := HwInputs.ST70_3_DM260_EB_Result_Data_64_bytes_1[36];
	PlcInputs.ST70_3_DM260_EB_Result_Data_64_bytes_1[37] := HwInputs.ST70_3_DM260_EB_Result_Data_64_bytes_1[37];
	PlcInputs.ST70_3_DM260_EB_Result_Data_64_bytes_1[38] := HwInputs.ST70_3_DM260_EB_Result_Data_64_bytes_1[38];
	PlcInputs.ST70_3_DM260_EB_Result_Data_64_bytes_1[39] := HwInputs.ST70_3_DM260_EB_Result_Data_64_bytes_1[39];
	PlcInputs.ST70_3_DM260_EB_Result_Data_64_bytes_1[40] := HwInputs.ST70_3_DM260_EB_Result_Data_64_bytes_1[40];
	PlcInputs.ST70_3_DM260_EB_Result_Data_64_bytes_1[41] := HwInputs.ST70_3_DM260_EB_Result_Data_64_bytes_1[41];
	PlcInputs.ST70_3_DM260_EB_Result_Data_64_bytes_1[42] := HwInputs.ST70_3_DM260_EB_Result_Data_64_bytes_1[42];
	PlcInputs.ST70_3_DM260_EB_Result_Data_64_bytes_1[43] := HwInputs.ST70_3_DM260_EB_Result_Data_64_bytes_1[43];
	PlcInputs.ST70_3_DM260_EB_Result_Data_64_bytes_1[44] := HwInputs.ST70_3_DM260_EB_Result_Data_64_bytes_1[44];
	PlcInputs.ST70_3_DM260_EB_Result_Data_64_bytes_1[45] := HwInputs.ST70_3_DM260_EB_Result_Data_64_bytes_1[45];
	PlcInputs.ST70_3_DM260_EB_Result_Data_64_bytes_1[46] := HwInputs.ST70_3_DM260_EB_Result_Data_64_bytes_1[46];
	PlcInputs.ST70_3_DM260_EB_Result_Data_64_bytes_1[47] := HwInputs.ST70_3_DM260_EB_Result_Data_64_bytes_1[47];
	PlcInputs.ST70_3_DM260_EB_Result_Data_64_bytes_1[48] := HwInputs.ST70_3_DM260_EB_Result_Data_64_bytes_1[48];
	PlcInputs.ST70_3_DM260_EB_Result_Data_64_bytes_1[49] := HwInputs.ST70_3_DM260_EB_Result_Data_64_bytes_1[49];
	PlcInputs.ST70_3_DM260_EB_Result_Data_64_bytes_1[50] := HwInputs.ST70_3_DM260_EB_Result_Data_64_bytes_1[50];
	PlcInputs.ST70_3_DM260_EB_Result_Data_64_bytes_1[51] := HwInputs.ST70_3_DM260_EB_Result_Data_64_bytes_1[51];
	PlcInputs.ST70_3_DM260_EB_Result_Data_64_bytes_1[52] := HwInputs.ST70_3_DM260_EB_Result_Data_64_bytes_1[52];
	PlcInputs.ST70_3_DM260_EB_Result_Data_64_bytes_1[53] := HwInputs.ST70_3_DM260_EB_Result_Data_64_bytes_1[53];
	PlcInputs.ST70_3_DM260_EB_Result_Data_64_bytes_1[54] := HwInputs.ST70_3_DM260_EB_Result_Data_64_bytes_1[54];
	PlcInputs.ST70_3_DM260_EB_Result_Data_64_bytes_1[55] := HwInputs.ST70_3_DM260_EB_Result_Data_64_bytes_1[55];
	PlcInputs.ST70_3_DM260_EB_Result_Data_64_bytes_1[56] := HwInputs.ST70_3_DM260_EB_Result_Data_64_bytes_1[56];
	PlcInputs.ST70_3_DM260_EB_Result_Data_64_bytes_1[57] := HwInputs.ST70_3_DM260_EB_Result_Data_64_bytes_1[57];
	PlcInputs.ST70_3_DM260_EB_Result_Data_64_bytes_1[58] := HwInputs.ST70_3_DM260_EB_Result_Data_64_bytes_1[58];
	PlcInputs.ST70_3_DM260_EB_Result_Data_64_bytes_1[59] := HwInputs.ST70_3_DM260_EB_Result_Data_64_bytes_1[59];
	PlcInputs.ST70_3_DM260_EB_Result_Data_64_bytes_1[60] := HwInputs.ST70_3_DM260_EB_Result_Data_64_bytes_1[60];
	PlcInputs.ST70_3_DM260_EB_Result_Data_64_bytes_1[61] := HwInputs.ST70_3_DM260_EB_Result_Data_64_bytes_1[61];
	PlcInputs.ST70_3_DM260_EB_Result_Data_64_bytes_1[62] := HwInputs.ST70_3_DM260_EB_Result_Data_64_bytes_1[62];
	PlcInputs.ST70_3_DM260_EB_Result_Data_64_bytes_1[63] := HwInputs.ST70_3_DM260_EB_Result_Data_64_bytes_1[63];
	PlcInputs.ST70_3_DM260_EB_Result_Data_64_bytes_1[64] := HwInputs.ST70_3_DM260_EB_Result_Data_64_bytes_1[64];
	PlcInputs.ST70_3_DM260_EB_Result_Data_64_bytes_1[65] := HwInputs.ST70_3_DM260_EB_Result_Data_64_bytes_1[65];
	PlcInputs.ST70_3_DM260_EB_Result_Data_64_bytes_1[66] := HwInputs.ST70_3_DM260_EB_Result_Data_64_bytes_1[66];
	PlcInputs.ST70_3_DM260_EB_Result_Data_64_bytes_1[67] := HwInputs.ST70_3_DM260_EB_Result_Data_64_bytes_1[67];
	PlcInputs.ST70_3_DM260_EB_Result_Data_64_bytes_1[68] := HwInputs.ST70_3_DM260_EB_Result_Data_64_bytes_1[68];
	PlcInputs.ST70_3_DM260_EB_Result_Data_64_bytes_1[69] := HwInputs.ST70_3_DM260_EB_Result_Data_64_bytes_1[69];
	PlcInputs.ST70_3_DM260_EB_Result_Data_64_bytes_1[70] := HwInputs.ST70_3_DM260_EB_Result_Data_64_bytes_1[70];
	PlcInputs.ST70_3_DM260_EB_Result_Data_64_bytes_1[71] := HwInputs.ST70_3_DM260_EB_Result_Data_64_bytes_1[71];
END_FUNCTION
